// TIA Portal V17 program export: 2 tag tables, 0 data types, 1 data blocks, 3 code blocks (in call order from the OBs), 0 instance data blocks

VAR_GLOBAL   // PLC tag table "Default tag table"
   Clock_Byte AT %MB0 : Byte;
   Clock_10Hz AT %M0.0 : Bool;
   Clock_5Hz AT %M0.1 : Bool;
   "Clock_2.5Hz" AT %M0.2 : Bool;
   Clock_2Hz AT %M0.3 : Bool;
   "Clock_1.25Hz" AT %M0.4 : Bool;
   Clock_1Hz AT %M0.5 : Bool;
   "Clock_0.625Hz" AT %M0.6 : Bool;
   "Clock_0.5Hz" AT %M0.7 : Bool;
   System_Byte AT %MB1 : Byte;
   FirstScan AT %M1.0 : Bool;
   DiagStatusUpdate AT %M1.1 : Bool;
   AlwaysTRUE AT %M1.2 : Bool;
   AlwaysFALSE AT %M1.3 : Bool;
   "System_Byte(1)" AT %MB1 : Byte;
END_VAR

VAR_GLOBAL   // PLC tag table "IO"
   IB_0 AT %IB0 : Byte;
   IB_1 AT %IB1 : Byte;
   QB_0 AT %QB0 : Byte;
   QB_1 AT %QB1 : Byte;
END_VAR

DATA_BLOCK "Data_block_1"   // DB1
{ S7_Optimized_Access := 'TRUE' }
VERSION : 0.1
// stored: AutoNumber true, DBAccessibleFromOPCUA true, IsOnlyStoredInLoadMemory false, IsRetainMemResEnabled false, IsWriteProtectedInAS false, MemoryReserve 100
   VAR
      aliveUDINT : UDInt;
   END_VAR
BEGIN
END_DATA_BLOCK

ORGANIZATION_BLOCK "Main"   // OB1, LAD, ProgramCycle
TITLE = "Main Program Sweep (Cycle)"
{ S7_Optimized_Access := 'TRUE' }
VERSION : 0.1
// stored: AutoNumber true, IsIECCheckEnabled false, SetENOAutomatically false
   VAR_INPUT
      Initial_Call : Bool;   // Initial call of this OB
      Remanence : Bool;   // =True, if remanent data are available
   END_VAR
BEGIN
END_ORGANIZATION_BLOCK

FUNCTION "FC_NormScaleAnalogInput" : Void   // FC1, LAD
{ S7_Optimized_Access := 'TRUE' }
VERSION : 0.1
// stored: AutoNumber true, IsIECCheckEnabled false, SetENOAutomatically false, UDAEnableTagReadback false
   VAR_INPUT
      AnalogInput : Int;   // Analog input [value 0 - 27648]
      minScaledValue : Real;   // lower value for scaled value Real
      maxScaledValue : Real;   // Upper value for scaled value Real
   END_VAR
   VAR_OUTPUT
      AnalogInputReal : Real;   // Scaled analog value Real
   END_VAR
   VAR_TEMP
      normAnalogValue : Real;
   END_VAR
   VAR CONSTANT
      LOWERINT : Int := 0;
      UPPERINT : Int := 27648;
   END_VAR
BEGIN

REGION Network 1
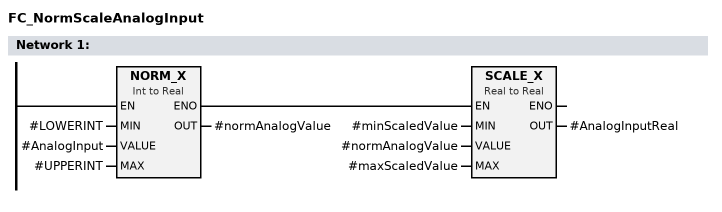
   RUNG wire#powerrail
      { S7_Templates := "[SrcType := Int, DestType := Real]" } Normalize(min := #LOWERINT, value := #AnalogInput, max := #UPPERINT, out => #normAnalogValue)
      { S7_Templates := "[SrcType := Real, DestType := Real]" } Scale(min := #minScaledValue, value := #normAnalogValue, max := #maxScaledValue, out => #AnalogInputReal)
   END_RUNG
   // the same network as SCL:
   #normAnalogValue := NORM_X(MIN := #LOWERINT, VALUE := #AnalogInput, MAX := #UPPERINT);
   #AnalogInputReal := SCALE_X(MIN := #minScaledValue, VALUE := #normAnalogValue, MAX := #maxScaledValue);
END_REGION
END_FUNCTION

FUNCTION "Alive" : Void
TITLE = Alive function
{ S7_Optimized_Access := 'TRUE' }
AUTHOR : MIGA
FAMILY : UCN
VERSION : 0.4
//This is a comment to the function
   VAR_IN_OUT 
      aliveInt : UDInt;
   END_VAR


BEGIN
	(*
	DETTE PROJEKT TILHØRER NU DANMARKS STØRSTE SPILER - - - HUSK AT LIKE OG SUBCRIBE TIL AdruEma PÅ GITHUB - - -
	This is a comment
	This FC is now also a type in libraries
	Vi er her stadig auta-csd-s22
	*)
	
	#aliveInt := #aliveInt + 1;
	IF #aliveInt > 1000 THEN
	    #aliveInt := 0;
	END_IF;
END_FUNCTION
